// TIA Portal V20 export
// export: Created 2025-12-01T14:57:22.4412966Z, ExportSetting None, DisplayName Totally Integrated Automation Portal, DisplayVersion V20 Update 3, DisplayName TIA Portal Openness, DisplayVersion V20 Update 3, DisplayName TIA Portal Version Control Interface, DisplayVersion V20 Update 3, DisplayName STEP 7 Professional, DisplayVersion V20 Update 3, DisplayName STEP 7 Safety, DisplayVersion V20 Update 2, DisplayName WinCC Basic/Comfort/Advanced, DisplayVersion V20 Update 3, DisplayName WinCC Professional, DisplayVersion V20 Update 3, DisplayName WinCC Unified, DisplayVersion V20 Update 3
DATA_BLOCK "DB915_Sinoptico_Ndd"   // DB915
{ S7_Optimized_Access := 'FALSE'; DB_Accessible_From_OPC_UA := 'FALSE' }
// stored: AutoNumber false, DBAccessibleFromOPCUA false
   VAR
      NDD : Array[1..10] of Struct
         Linea { S7_SetPoint := 'True'} : Array[0..9] of "UDT_HMI_LineaPotencia";
      END_STRUCT;
   END_VAR
BEGIN
END_DATA_BLOCK
